INTERFACE I_ControlType

METHOD Joystick
VAR_INPUT
	bSwitch : BOOL;
	bActive : BOOL;
END_VAR
END_METHOD

METHOD Mode
VAR_INPUT
	eCurrentMode : E_Mode;
END_VAR
END_METHOD

METHOD Status
VAR_INPUT
	eStatus : E_Status;
END_VAR
END_METHOD

END_INTERFACE

(* stored: Version 1.1.0.1, ProductVersion 3.1.4024.12
   Itf I_ControlType: Id {c3d0b8cd-a2e5-4cf6-a7af-6729a2c0238a}
   Method Joystick: Id {092f3369-1f84-408c-9be7-56d5e5c3ae50}
   Method Mode: Id {8ea05e7a-e48a-4272-8f39-4382aec6a3a4}
   Method Status: Id {22bdb8b7-ddbe-4802-948f-92f2936fd6a5} *)
